FUNCTION_BLOCK BIT_TO_WORD_V0
VAR_INPUT
	bit0:BIT;
	bit1:BIT;
	bit2:BIT;
	bit3:BIT;
	bit4:BIT;
	bit5:BIT;
	bit6:BIT;
	bit7:BIT;
	bit8:BIT;
	bit9:BIT;
	bit10:BIT;
	bit11:BIT;
	bit12:BIT;
	bit13:BIT;
	bit14:BIT;
	bit15:BIT;
END_VAR
VAR_OUTPUT
	Word_out:WORD;
END_VAR
VAR
END_VAR
VAR // added by the converter: edge detectors and wires of the graphical bodies
    _w1, _w2, _w3, _w4, _w5, _w6, _w7, _w8, _w9, _w10, _w11, _w12, _w13, _w14, _w15 : ANY;
END_VAR

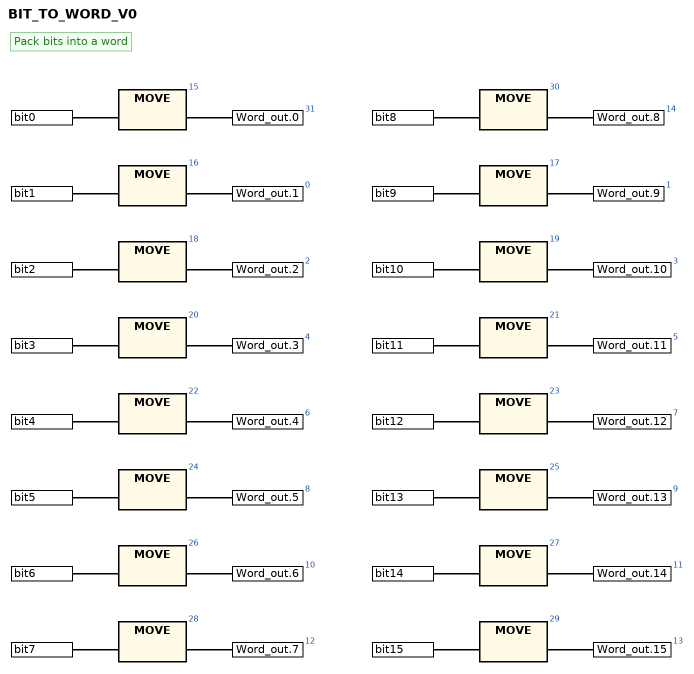
Word_out.1 := _w1;
Word_out.9 := _w2;
Word_out.2 := _w3;
Word_out.10 := _w4;
Word_out.3 := _w5;
Word_out.11 := _w6;
Word_out.4 := _w7;
Word_out.12 := _w8;
Word_out.5 := _w9;
Word_out.13 := _w10;
Word_out.6 := _w11;
Word_out.14 := _w12;
Word_out.7 := _w13;
Word_out.15 := _w14;
Word_out.8 := _w15;
// Pack bits into a word
_w1 := bit1;
_w2 := bit9;
_w3 := bit2;
_w4 := bit10;
_w5 := bit3;
_w6 := bit11;
_w7 := bit4;
_w8 := bit12;
_w9 := bit5;
_w10 := bit13;
_w11 := bit6;
_w12 := bit14;
_w13 := bit7;
_w14 := bit15;
_w15 := bit8;
Word_out.0 := bit0;

END_FUNCTION_BLOCK

(* stored: Version 1.1.0.1, ProductVersion 3.1.4024.0
   POU BIT_TO_WORD_V0: Id {2c3ea628-83f8-4386-bfed-caf9960d70f3}, SpecialFunc None *)
